FUNCTION_BLOCK E_SWITCH (* Switching (demultiplexing) an event based on boolean input G *)
  (* Standard: 61499-1 Annex A; Description: Copyright (c) 2017 fortiss GmbH This program and the accompanying materials are made available under the terms of the Eclipse Public License 2.0 which is available at https://www.eclipse.org/legal/epl-2.0/ SPDX-License-Identifier: EPL-2.0 *)
  (* Version 1.0, 2017-09-21, Alois Zoitl, fortiss GmbH, initial API and implementation and/or initial documentation *)
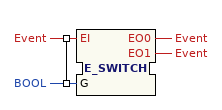
  EVENT_INPUT
    EI WITH G; (* Event Input *)
  END_EVENT
  EVENT_OUTPUT
    EO0; (* Output, switched from EI when G=0 *)
    EO1; (* Output, switched from EI when G=1 *)
  END_EVENT
  VAR_INPUT
    G : BOOL; (* Switch EI to EI0 when G=0, to EI1 when G=1 *)
  END_VAR
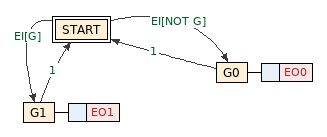
  EC_STATES
    START; (* Initial State *)
    G0 : -> EO0; (* Issue EO0 when EI arrives with G=0 *)
    G1 : -> EO1; (* Issue EO1 when EI arrives with G=1 *)
  END_STATES
  EC_TRANSITIONS
    G0 TO START := 1;
    G1 TO START := 1;
    START TO G0 := EI[NOT G];
    START TO G1 := EI[G];
  END_TRANSITIONS
END_FUNCTION_BLOCK
